(* Logix 5000 project; controller cal1615 1756-L62 rev 20.11; software revision 20.05; part 51 of 82 *)
(* tags used below, declared in another part *)
   FAULT : BOOL;   // Fault AFI
   HMI : BOOL;   // AFI HMI
   p01r09_pb_global_reset : BOOL;   // System Modes PB: Global Fault Reset
   p23_ai_os_gap_dint : DINT;
   p23_ai_os_masked_gap : REAL;
   p23_ai_servo_os_position : REAL;   // Impreg Inputs Servo Operator Side Position
   p23_ai_servo_os_torque : REAL;   // Impreg Inputs Servo Operator Side Torque
   p23_ao_selected_speed : REAL;   // Impreg Metering Roll VFD Selected Speed
   p23_ao_servo_ds_jog_vel_cmd : REAL;   // Impreg Servo Drive Side Jog Velocity Command [in/sec]
   p23_ao_servo_ds_position_cmd : REAL;   // Impreg Servo Drive Side Position Command
   p23_ao_servo_ds_velocity_cmd : REAL;   // Impreg Servo Drive Side Velocity Command
   p23_ao_servo_ds_zero_offset : REAL;   // Impreg Analog Outputs Drive Side Servo Position Offset
   p23_ao_servo_os_jog_vel_cmd : REAL;   // Impreg Servo Operator Side Jog Velocity Command [in/sec]
   p23_ao_servo_os_position_cmd : REAL;   // Impreg Servo Operator Side Position Command
   p23_ao_servo_os_velocity_cmd : REAL;   // Impreg Servo Operator Side Velocity Command
   p23_ao_servo_os_zero_offset : REAL;   // Impreg Analog Outputs Drive Operator Side Servo Position Offset
   p23_ao_supply_selected_speed : REAL;   // Impreg Supply VFD Selected Speed
   p23_cpr_gear_ratio : REAL;
   p23_cpr_roll_diameter_ft : REAL;
   p23_cpr_speed_to_vfd : SYS_SPEED_TO_VFD;   // Impreg Outputs Speed to Impreg Pick Up Roll VFD
   p23_di_impreg_tank_up : BOOL;   // Input Impreg Dip Tank Up
   p23_di_metering_roll : acs800_di_normal;   // Impreg Digital Inputs Metering Roll VFD
   p23_di_servo_ds : servo_di;   // Impreg Digital Inputs Servo Drive Side
   p23_di_servo_os : servo_di;   // Impreg Digital Inputs Servo Operator Side
   p23_di_supply : acs800_di_normal;   // Impreg Supply VFD VFD Inputs
   p23_di_tank_level_high : BOOL;   // Impreg Input Dip Impreg Level High
   p23_di_tank_level_low : BOOL;   // Impreg Input Dip Impreg Level Low
   p23_di_though_level_low : BOOL;   // Impreg Input Dip Impreg Through Level Low
   p23_dint_to_hmi : DINT[17];   // Impreg Dint to HMI
   p23_do_enable_impreg_exhaust_fan : BOOL;   // Impreg Enclosure Digital Output Exhaust Fan Enable
   p23_do_enable_impreg_supply_fan : BOOL;   // Impreg Enclosure Digital Output Supply Fan Enable
   p23_do_impreg : acs800_do_normal;   // Impreg Digital Outputs VFD
   p23_do_impreg_nip_close : BOOL;   // Impreg Digital Output Impreg Nip close
   p23_do_servo_ds : servo_do;   // Impreg Digital Outputs Drive Side Servo
   p23_do_servo_os : servo_do;   // Impreg Digital Outputs Operator Side Servo
   p23_do_Spring : acs800_do_normal;
   p23_do_supply : acs800_do_normal;   // Impreg Supply VFD] Outputs
   p23_servo_ds_error : SYS_ENC_WITH_ZERO_BIT;   // Impreg Dint to HMI Servo Drive Side Error
   p23_servo_ds_warning : SYS_ENC_WITH_ZERO_BIT;   // Impreg Dint to HMI Servo Drive Side Warning
   p23_servo_os_error : SYS_ENC_WITH_ZERO_BIT;   // Impreg Dint to HMI Servo Operator Side Error
   p23_spring_gear_ratio : REAL;
   p23_spring_roll_diameter_ft : REAL;
   p23_spring_speed_to_vfd : SYS_SPEED_TO_VFD;
   p23r01 : routine;   // Impreg Main
   p23r03 : routine;   // Impreg Inputs
   p23r03_timer_fault : TIMER[4];   // Impreg Inputs Timer Fault
   p23r03_timer_warning : TIMER[4];   // Impreg Inputs Timer Warning
   p23r04 : routine;   // Impreg Outputs
   p23r04_timer_fault : TIMER[4];   // Impreg Outputs Fault Delay
   p23r04_timer_warning : TIMER[4];   // Impreg Outputs Warning Delay
   p23r05 : routine;   // Impreg Dint to HMI
   p23r11_servo_not_ready : BOOL;   // Impreg Servo Operator Side Not Ready
   p23r11_servo_status_ab : BOOL;   // Impreg Servo Operator Side AB Status
   p23r11_servo_status_af : BOOL;   // Impreg Servo Operator Side AF Status
   p23r11_servo_status_bb : BOOL;   // Impreg Servo Operator Side BB Status
   p23r12_servo_not_ready : BOOL;   // Impreg Servo Drive Side Not Ready
   p23r12_servo_status_ab : BOOL;   // Impreg Servo Drive Side AB Status
   p23r12_servo_status_af : BOOL;   // Impreg Servo Drive Side AF Status
   p23r12_servo_status_bb : BOOL;   // Impreg Servo Drive Side BB Status
   p23r15_pid_tension_control : BOOL;   // Impreg Metering Roll VFD PID Wet Web Active
   p23r17_adjusted_speed : REAL;
(* P23_Impreg, continued *)

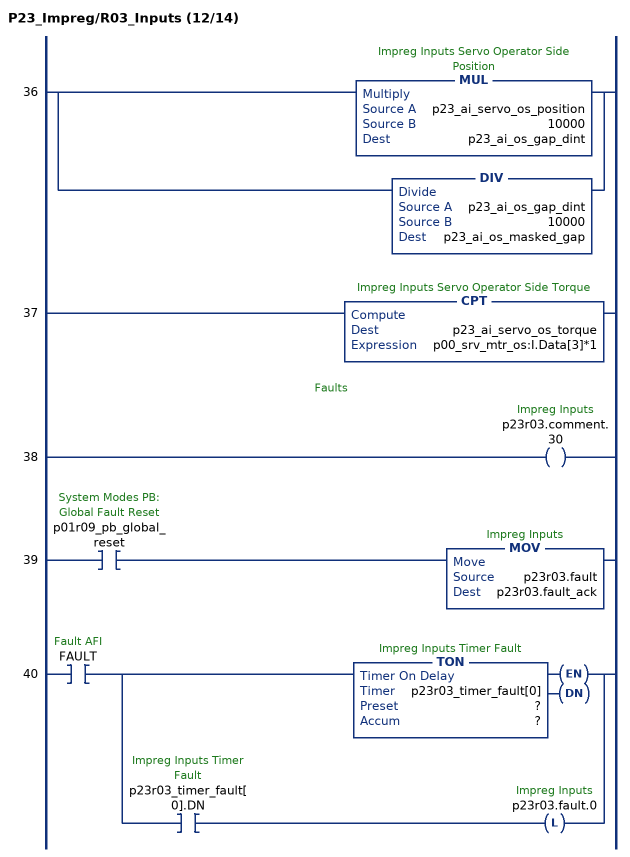
   [picture p993: P23_Impreg/R03_Inputs rungs 36-40]
   36: [MUL(p23_ai_servo_os_position,10000,p23_ai_os_gap_dint) ,DIV(p23_ai_os_gap_dint,10000,p23_ai_os_masked_gap) ];
   37: CPT(p23_ai_servo_os_torque,p00_srv_mtr_os:I.Data[3]*1);
   // Faults
   38: OTE(p23r03.comment.30);
   39: XIC(p01r09_pb_global_reset)MOV(p23r03.fault,p23r03.fault_ack);
   40: XIC(FAULT)[TON(p23r03_timer_fault[0],?,?) ,XIC(p23r03_timer_fault[0].DN) OTL(p23r03.fault.0) ];
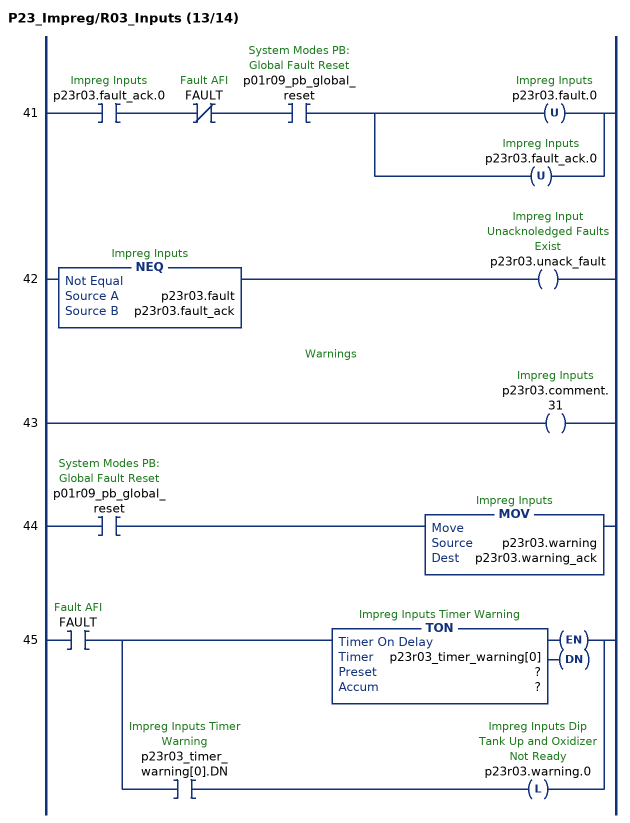
   41: XIC(p23r03.fault_ack.0)XIO(FAULT)XIC(p01r09_pb_global_reset)[OTU(p23r03.fault.0) ,OTU(p23r03.fault_ack.0) ];
   42: NEQ(p23r03.fault,p23r03.fault_ack)OTE(p23r03.unack_fault);
   // Warnings
   43: OTE(p23r03.comment.31);
   44: XIC(p01r09_pb_global_reset)MOV(p23r03.warning,p23r03.warning_ack);
   45: XIC(FAULT)[TON(p23r03_timer_warning[0],?,?) ,XIC(p23r03_timer_warning[0].DN) OTL(p23r03.warning.0) ];
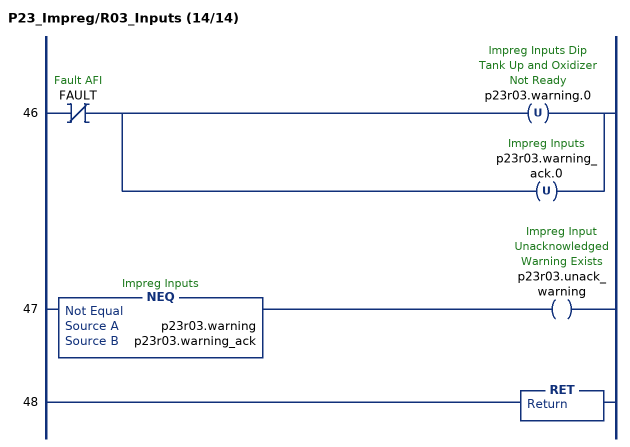
   46: XIO(FAULT)[OTU(p23r03.warning.0) ,OTU(p23r03.warning_ack.0) ];
   47: NEQ(p23r03.warning,p23r03.warning_ack)OTE(p23r03.unack_warning);
   48: RET();
END_ROUTINE

ROUTINE R04_Outputs   (* ladder *)
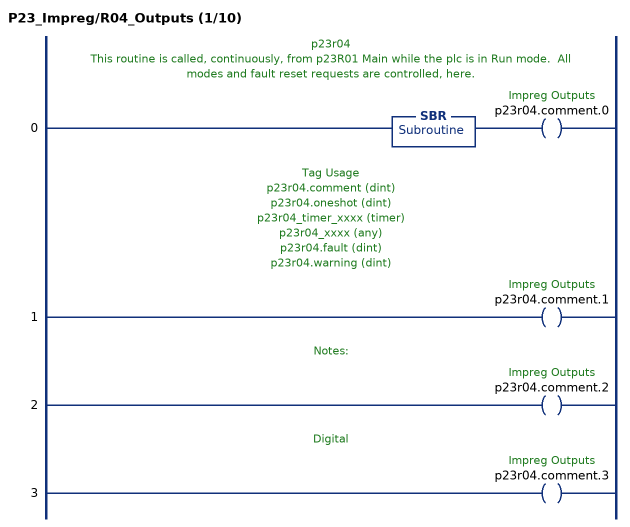
   // p23r04
   // This routine is called, continuously, from p23R01 Main while the plc is in Run mode.  All modes and fault reset requests are controlled, here.
   0: SBR()OTE(p23r04.comment.0);
   // Tag Usage
   // p23r04.comment (dint)
   // p23r04.oneshot (dint)
   // p23r04_timer_xxxx (timer)
   // p23r04_xxxx (any)
   // p23r04.fault (dint)
   // p23r04.warning (dint)
   1: OTE(p23r04.comment.1);
   // Notes:
   2: OTE(p23r04.comment.2);
   // Digital
   3: OTE(p23r04.comment.3);
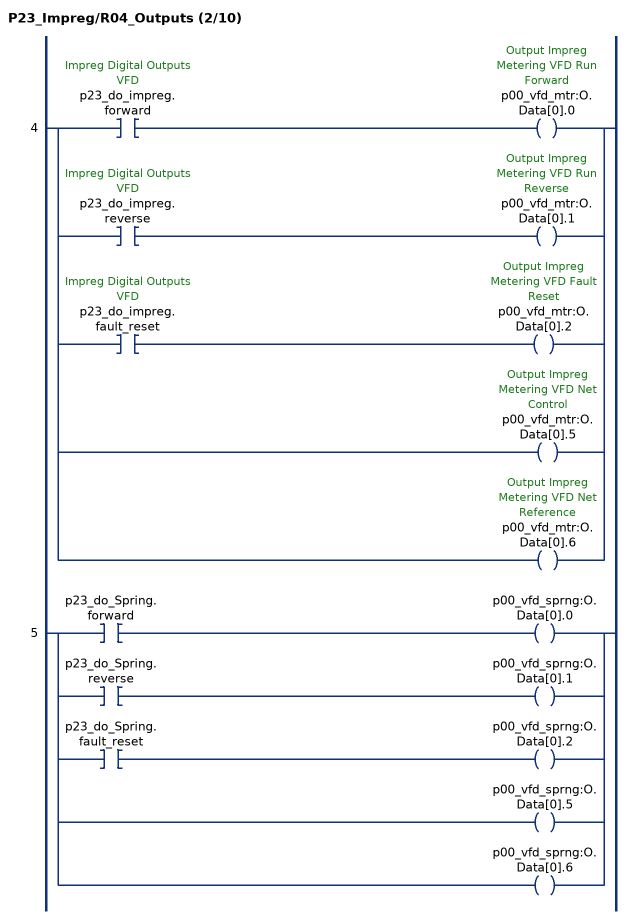
   4: [XIC(p23_do_impreg.forward) OTE(p00_vfd_mtr:O.Data[0].0) ,XIC(p23_do_impreg.reverse) OTE(p00_vfd_mtr:O.Data[0].1) ,XIC(p23_do_impreg.fault_reset) OTE(p00_vfd_mtr:O.Data[0].2) ,OTE(p00_vfd_mtr:O.Data[0].5) ,OTE(p00_vfd_mtr:O.Data[0].6) ];
   5: [XIC(p23_do_Spring.forward) OTE(p00_vfd_sprng:O.Data[0].0) ,XIC(p23_do_Spring.reverse) OTE(p00_vfd_sprng:O.Data[0].1) ,XIC(p23_do_Spring.fault_reset) OTE(p00_vfd_sprng:O.Data[0].2) ,OTE(p00_vfd_sprng:O.Data[0].5) ,OTE(p00_vfd_sprng:O.Data[0].6) ];
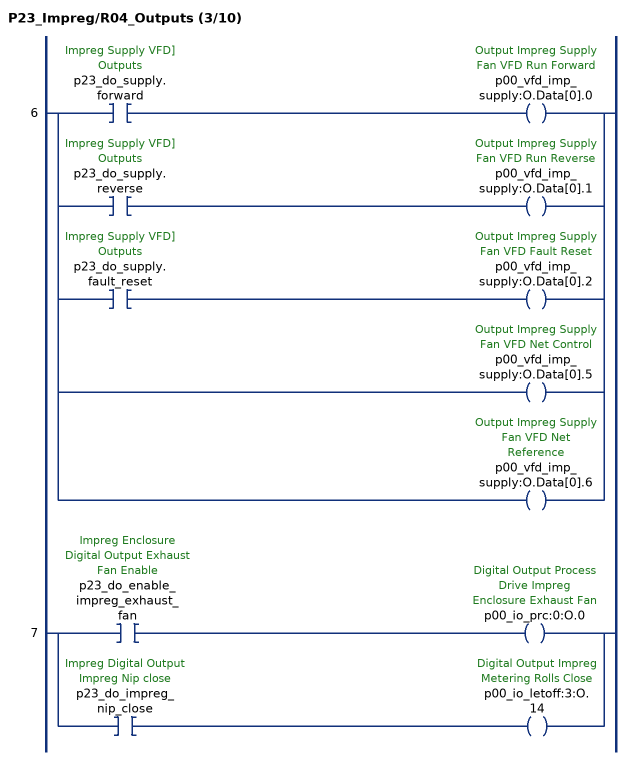
   6: [XIC(p23_do_supply.forward) OTE(p00_vfd_imp_supply:O.Data[0].0) ,XIC(p23_do_supply.reverse) OTE(p00_vfd_imp_supply:O.Data[0].1) ,XIC(p23_do_supply.fault_reset) OTE(p00_vfd_imp_supply:O.Data[0].2) ,OTE(p00_vfd_imp_supply:O.Data[0].5) ,OTE(p00_vfd_imp_supply:O.Data[0].6) ];
   7: [XIC(p23_do_enable_impreg_exhaust_fan) OTE(p00_io_prc:0:O.0) ,XIC(p23_do_impreg_nip_close) OTE(p00_io_letoff:3:O.14) ];
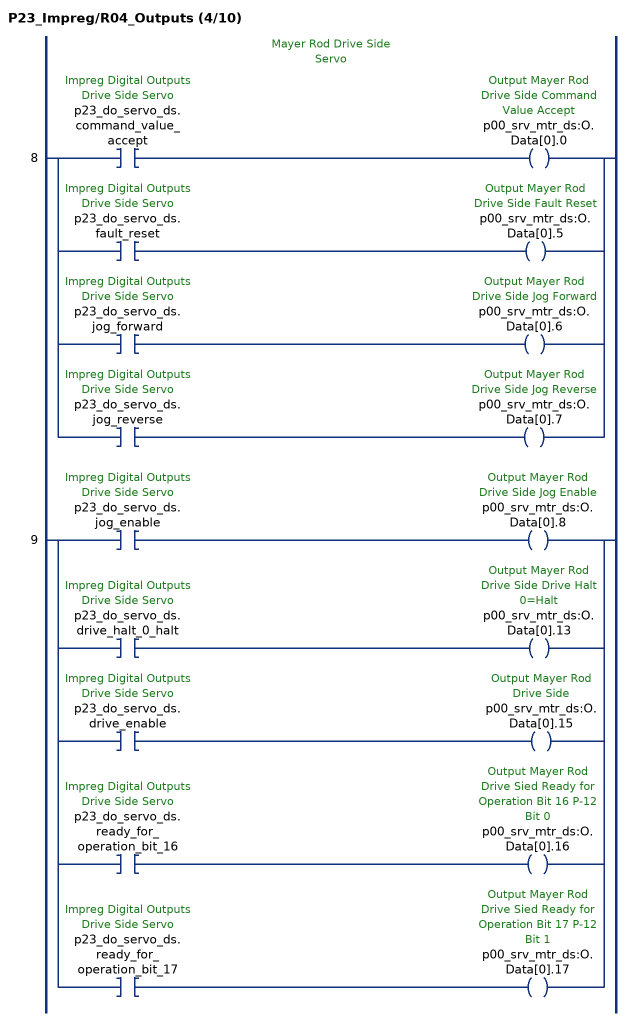
   // Mayer Rod Drive Side
   // Servo
   8: [XIC(p23_do_servo_ds.command_value_accept) OTE(p00_srv_mtr_ds:O.Data[0].0) ,XIC(p23_do_servo_ds.fault_reset) OTE(p00_srv_mtr_ds:O.Data[0].5) ,XIC(p23_do_servo_ds.jog_forward) OTE(p00_srv_mtr_ds:O.Data[0].6) ,XIC(p23_do_servo_ds.jog_reverse) OTE(p00_srv_mtr_ds:O.Data[0].7) ];
   9: [XIC(p23_do_servo_ds.jog_enable) OTE(p00_srv_mtr_ds:O.Data[0].8) ,XIC(p23_do_servo_ds.drive_halt_0_halt) OTE(p00_srv_mtr_ds:O.Data[0].13) ,XIC(p23_do_servo_ds.drive_enable) OTE(p00_srv_mtr_ds:O.Data[0].15) ,XIC(p23_do_servo_ds.ready_for_operation_bit_16) OTE(p00_srv_mtr_ds:O.Data[0].16) ,XIC(p23_do_servo_ds.ready_for_operation_bit_17) OTE(p00_srv_mtr_ds:O.Data[0].17) ];
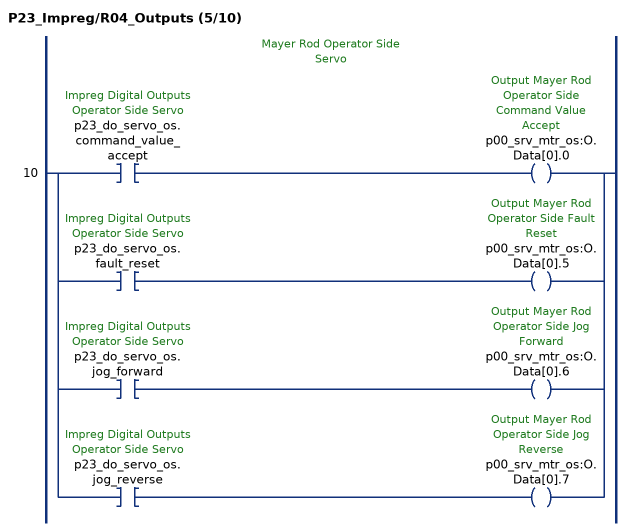
   // Mayer Rod Operator Side
   // Servo
   10: [XIC(p23_do_servo_os.command_value_accept) OTE(p00_srv_mtr_os:O.Data[0].0) ,XIC(p23_do_servo_os.fault_reset) OTE(p00_srv_mtr_os:O.Data[0].5) ,XIC(p23_do_servo_os.jog_forward) OTE(p00_srv_mtr_os:O.Data[0].6) ,XIC(p23_do_servo_os.jog_reverse) OTE(p00_srv_mtr_os:O.Data[0].7) ];
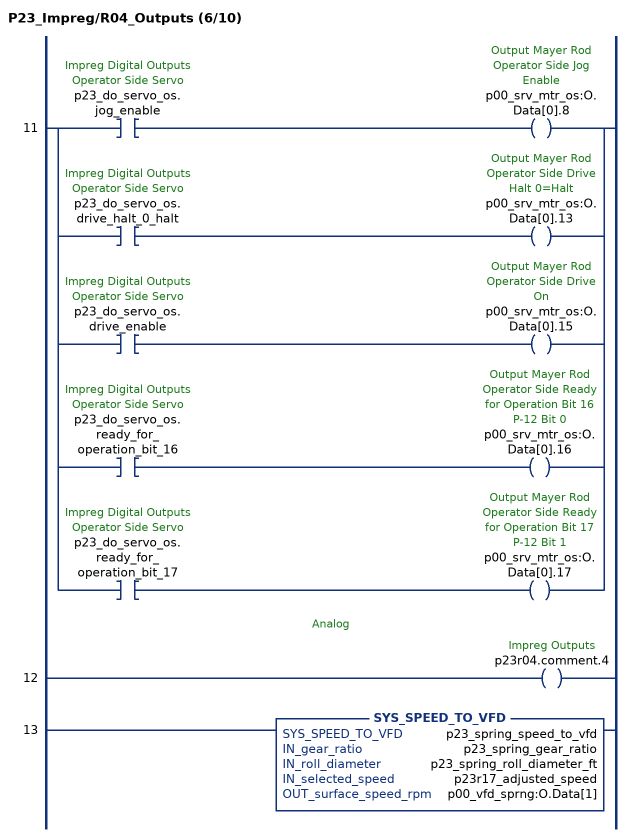
   11: [XIC(p23_do_servo_os.jog_enable) OTE(p00_srv_mtr_os:O.Data[0].8) ,XIC(p23_do_servo_os.drive_halt_0_halt) OTE(p00_srv_mtr_os:O.Data[0].13) ,XIC(p23_do_servo_os.drive_enable) OTE(p00_srv_mtr_os:O.Data[0].15) ,XIC(p23_do_servo_os.ready_for_operation_bit_16) OTE(p00_srv_mtr_os:O.Data[0].16) ,XIC(p23_do_servo_os.ready_for_operation_bit_17) OTE(p00_srv_mtr_os:O.Data[0].17) ];
   // Analog
   12: OTE(p23r04.comment.4);
   13: SYS_SPEED_TO_VFD(p23_spring_speed_to_vfd,p23_spring_gear_ratio,p23_spring_roll_diameter_ft,p23r17_adjusted_speed,p00_vfd_sprng:O.Data[1]);
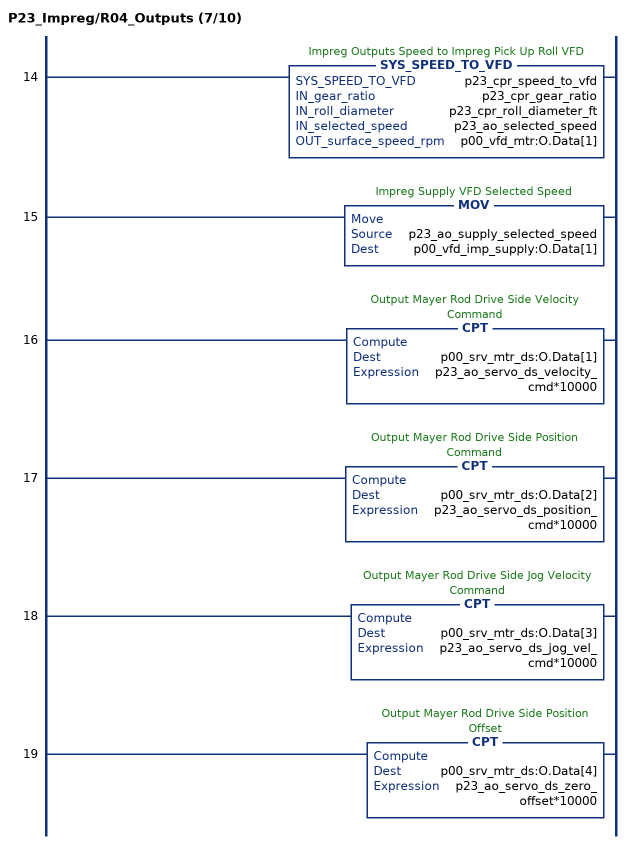
   14: SYS_SPEED_TO_VFD(p23_cpr_speed_to_vfd,p23_cpr_gear_ratio,p23_cpr_roll_diameter_ft,p23_ao_selected_speed,p00_vfd_mtr:O.Data[1]);
   15: MOV(p23_ao_supply_selected_speed,p00_vfd_imp_supply:O.Data[1]);
   16: CPT(p00_srv_mtr_ds:O.Data[1],p23_ao_servo_ds_velocity_cmd*10000);
   17: CPT(p00_srv_mtr_ds:O.Data[2],p23_ao_servo_ds_position_cmd*10000);
   18: CPT(p00_srv_mtr_ds:O.Data[3],p23_ao_servo_ds_jog_vel_cmd*10000);
   19: CPT(p00_srv_mtr_ds:O.Data[4],p23_ao_servo_ds_zero_offset*10000);
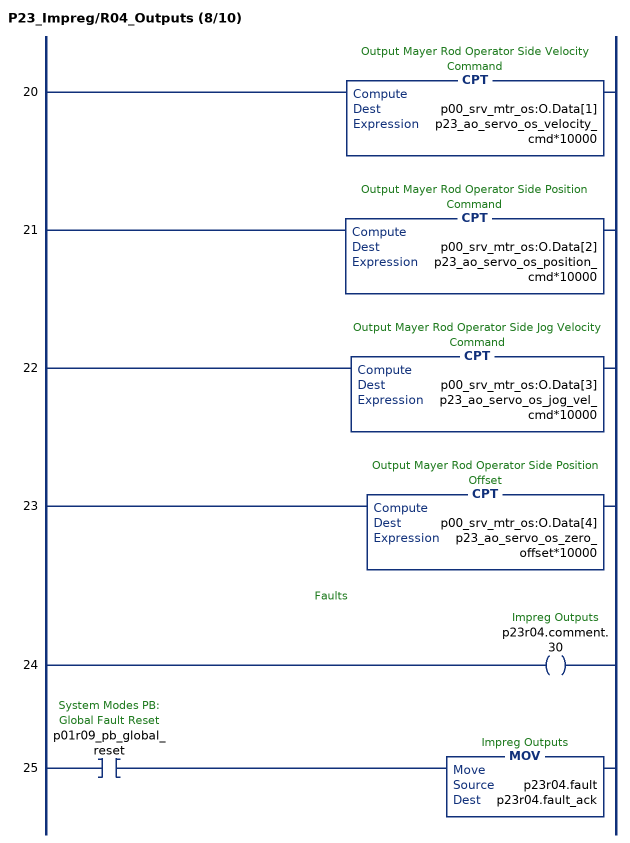
   20: CPT(p00_srv_mtr_os:O.Data[1],p23_ao_servo_os_velocity_cmd*10000);
   21: CPT(p00_srv_mtr_os:O.Data[2],p23_ao_servo_os_position_cmd*10000);
   22: CPT(p00_srv_mtr_os:O.Data[3],p23_ao_servo_os_jog_vel_cmd*10000);
   23: CPT(p00_srv_mtr_os:O.Data[4],p23_ao_servo_os_zero_offset*10000);
   // Faults
   24: OTE(p23r04.comment.30);
   25: XIC(p01r09_pb_global_reset)MOV(p23r04.fault,p23r04.fault_ack);
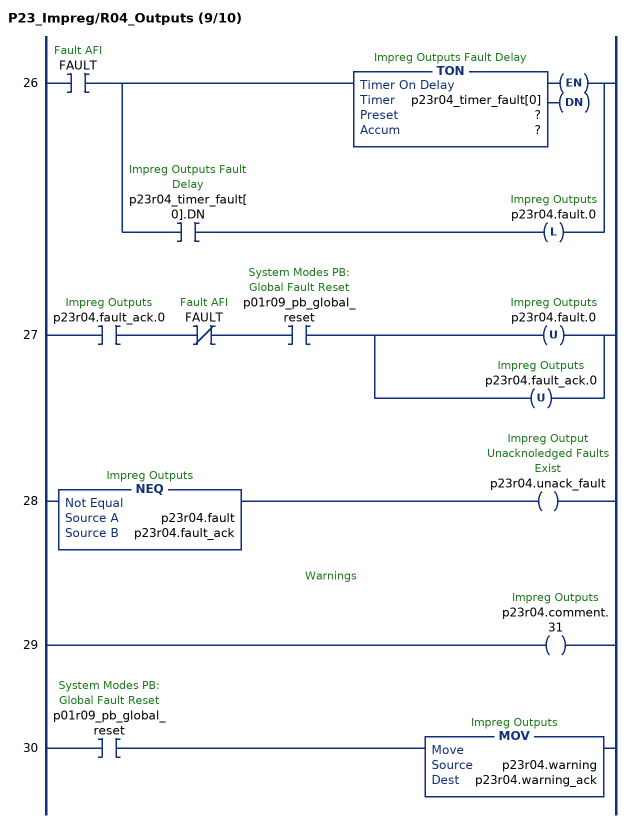
   26: XIC(FAULT)[TON(p23r04_timer_fault[0],?,?) ,XIC(p23r04_timer_fault[0].DN) OTL(p23r04.fault.0) ];
   27: XIC(p23r04.fault_ack.0)XIO(FAULT)XIC(p01r09_pb_global_reset)[OTU(p23r04.fault.0) ,OTU(p23r04.fault_ack.0) ];
   28: NEQ(p23r04.fault,p23r04.fault_ack)OTE(p23r04.unack_fault);
   // Warnings
   29: OTE(p23r04.comment.31);
   30: XIC(p01r09_pb_global_reset)MOV(p23r04.warning,p23r04.warning_ack);
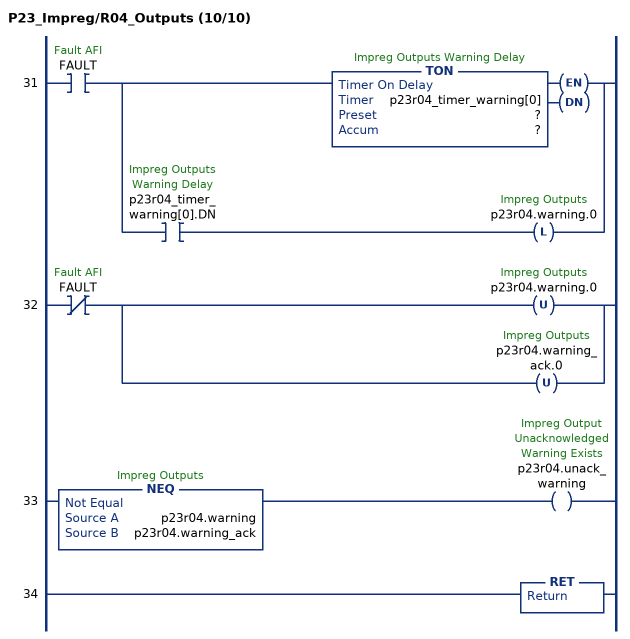
   31: XIC(FAULT)[TON(p23r04_timer_warning[0],?,?) ,XIC(p23r04_timer_warning[0].DN) OTL(p23r04.warning.0) ];
   32: XIO(FAULT)[OTU(p23r04.warning.0) ,OTU(p23r04.warning_ack.0) ];
   33: NEQ(p23r04.warning,p23r04.warning_ack)OTE(p23r04.unack_warning);
   34: RET();
END_ROUTINE

ROUTINE R05_Dint_to_HMI   (* ladder *)
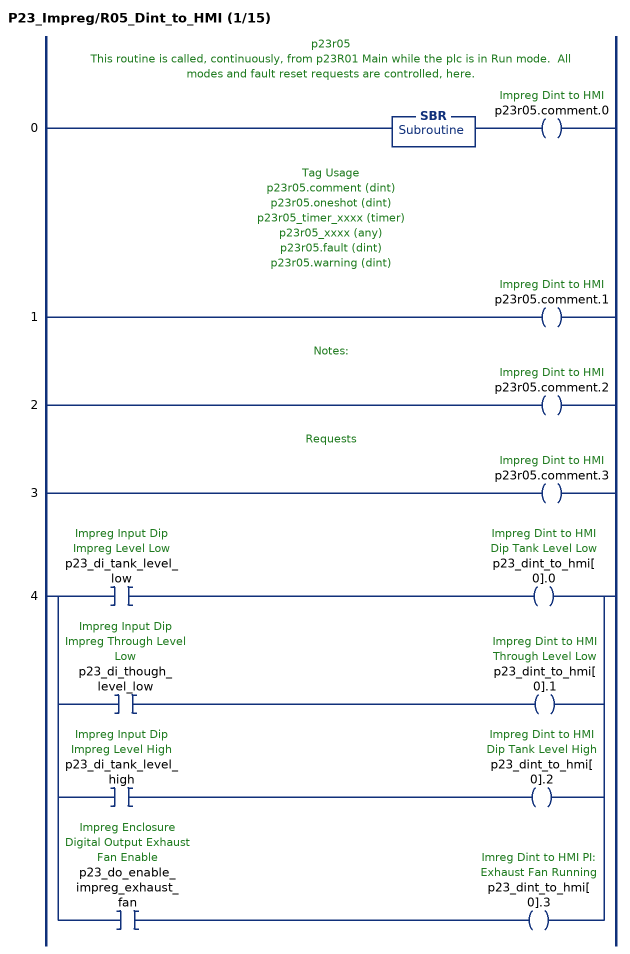
   // p23r05
   // This routine is called, continuously, from p23R01 Main while the plc is in Run mode.  All modes and fault reset requests are controlled, here.
   0: SBR()OTE(p23r05.comment.0);
   // Tag Usage
   // p23r05.comment (dint)
   // p23r05.oneshot (dint)
   // p23r05_timer_xxxx (timer)
   // p23r05_xxxx (any)
   // p23r05.fault (dint)
   // p23r05.warning (dint)
   1: OTE(p23r05.comment.1);
   // Notes:
   2: OTE(p23r05.comment.2);
   // Requests
   3: OTE(p23r05.comment.3);
   4: [XIC(p23_di_tank_level_low) OTE(p23_dint_to_hmi[0].0) ,XIC(p23_di_though_level_low) OTE(p23_dint_to_hmi[0].1) ,XIC(p23_di_tank_level_high) OTE(p23_dint_to_hmi[0].2) ,XIC(p23_do_enable_impreg_exhaust_fan) OTE(p23_dint_to_hmi[0].3) ];
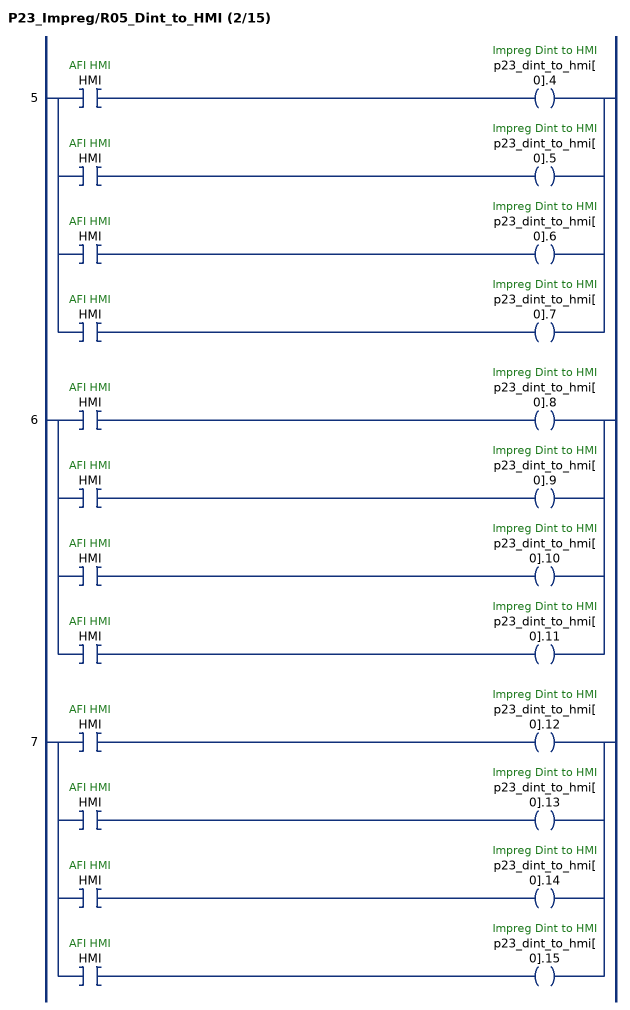
   5: [XIC(HMI) OTE(p23_dint_to_hmi[0].4) ,XIC(HMI) OTE(p23_dint_to_hmi[0].5) ,XIC(HMI) OTE(p23_dint_to_hmi[0].6) ,XIC(HMI) OTE(p23_dint_to_hmi[0].7) ];
   6: [XIC(HMI) OTE(p23_dint_to_hmi[0].8) ,XIC(HMI) OTE(p23_dint_to_hmi[0].9) ,XIC(HMI) OTE(p23_dint_to_hmi[0].10) ,XIC(HMI) OTE(p23_dint_to_hmi[0].11) ];
   7: [XIC(HMI) OTE(p23_dint_to_hmi[0].12) ,XIC(HMI) OTE(p23_dint_to_hmi[0].13) ,XIC(HMI) OTE(p23_dint_to_hmi[0].14) ,XIC(HMI) OTE(p23_dint_to_hmi[0].15) ];
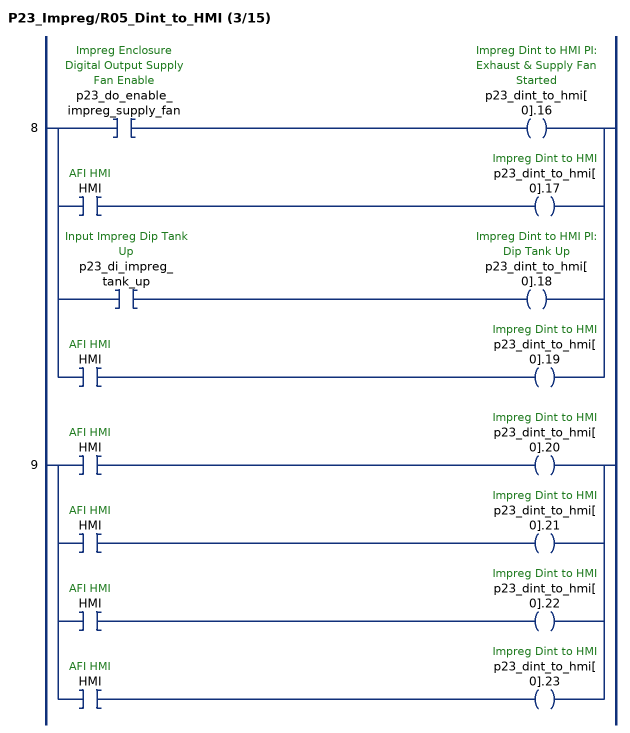
   8: [XIC(p23_do_enable_impreg_supply_fan) OTE(p23_dint_to_hmi[0].16) ,XIC(HMI) OTE(p23_dint_to_hmi[0].17) ,XIC(p23_di_impreg_tank_up) OTE(p23_dint_to_hmi[0].18) ,XIC(HMI) OTE(p23_dint_to_hmi[0].19) ];
   9: [XIC(HMI) OTE(p23_dint_to_hmi[0].20) ,XIC(HMI) OTE(p23_dint_to_hmi[0].21) ,XIC(HMI) OTE(p23_dint_to_hmi[0].22) ,XIC(HMI) OTE(p23_dint_to_hmi[0].23) ];
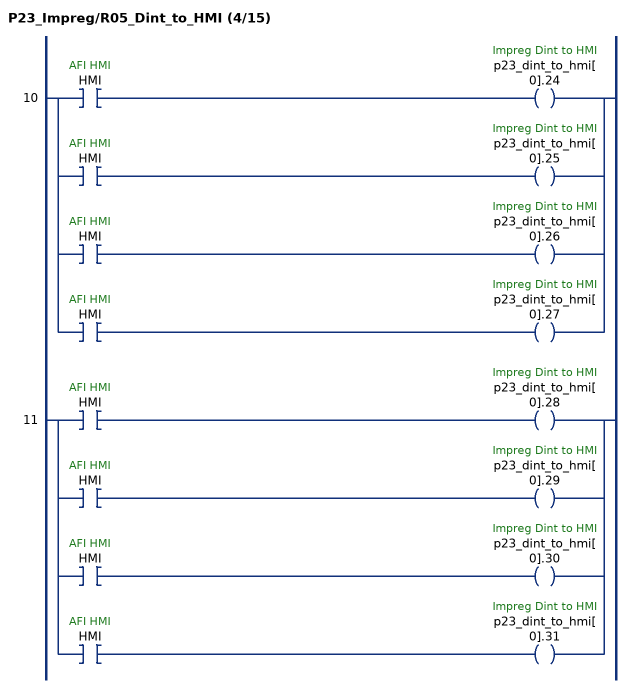
   10: [XIC(HMI) OTE(p23_dint_to_hmi[0].24) ,XIC(HMI) OTE(p23_dint_to_hmi[0].25) ,XIC(HMI) OTE(p23_dint_to_hmi[0].26) ,XIC(HMI) OTE(p23_dint_to_hmi[0].27) ];
   11: [XIC(HMI) OTE(p23_dint_to_hmi[0].28) ,XIC(HMI) OTE(p23_dint_to_hmi[0].29) ,XIC(HMI) OTE(p23_dint_to_hmi[0].30) ,XIC(HMI) OTE(p23_dint_to_hmi[0].31) ];
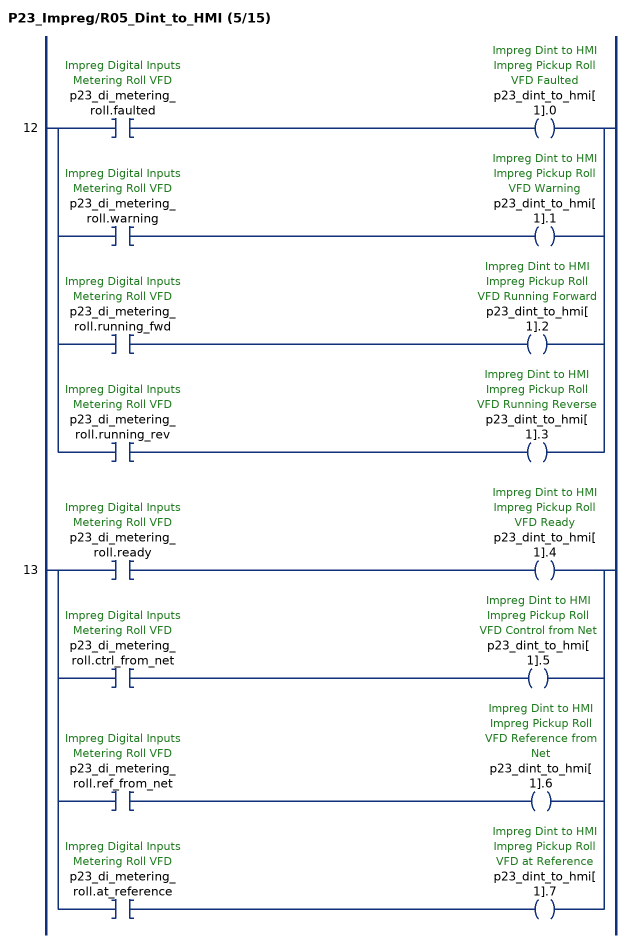
   12: [XIC(p23_di_metering_roll.faulted) OTE(p23_dint_to_hmi[1].0) ,XIC(p23_di_metering_roll.warning) OTE(p23_dint_to_hmi[1].1) ,XIC(p23_di_metering_roll.running_fwd) OTE(p23_dint_to_hmi[1].2) ,XIC(p23_di_metering_roll.running_rev) OTE(p23_dint_to_hmi[1].3) ];
   13: [XIC(p23_di_metering_roll.ready) OTE(p23_dint_to_hmi[1].4) ,XIC(p23_di_metering_roll.ctrl_from_net) OTE(p23_dint_to_hmi[1].5) ,XIC(p23_di_metering_roll.ref_from_net) OTE(p23_dint_to_hmi[1].6) ,XIC(p23_di_metering_roll.at_reference) OTE(p23_dint_to_hmi[1].7) ];
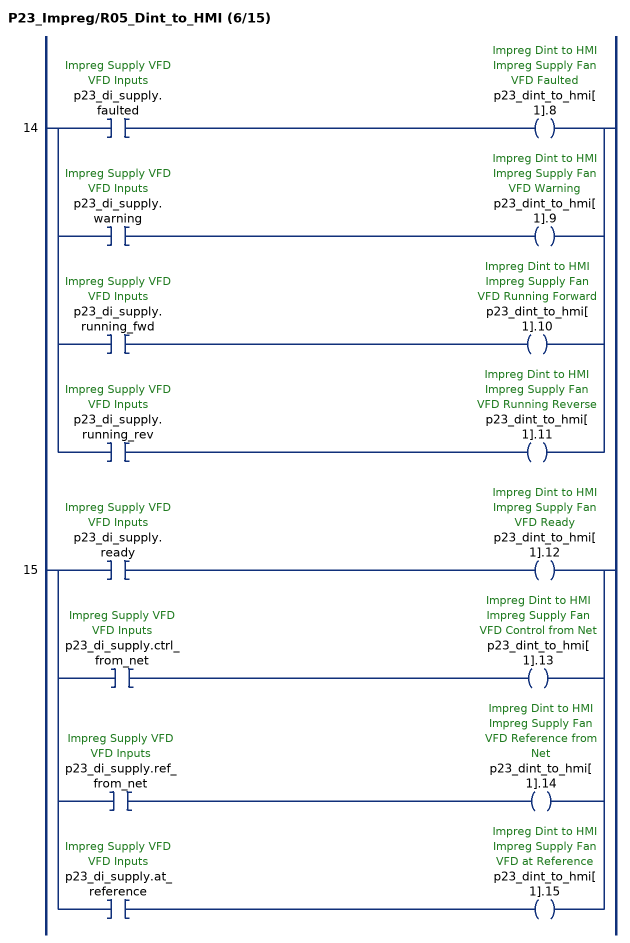
   14: [XIC(p23_di_supply.faulted) OTE(p23_dint_to_hmi[1].8) ,XIC(p23_di_supply.warning) OTE(p23_dint_to_hmi[1].9) ,XIC(p23_di_supply.running_fwd) OTE(p23_dint_to_hmi[1].10) ,XIC(p23_di_supply.running_rev) OTE(p23_dint_to_hmi[1].11) ];
   15: [XIC(p23_di_supply.ready) OTE(p23_dint_to_hmi[1].12) ,XIC(p23_di_supply.ctrl_from_net) OTE(p23_dint_to_hmi[1].13) ,XIC(p23_di_supply.ref_from_net) OTE(p23_dint_to_hmi[1].14) ,XIC(p23_di_supply.at_reference) OTE(p23_dint_to_hmi[1].15) ];
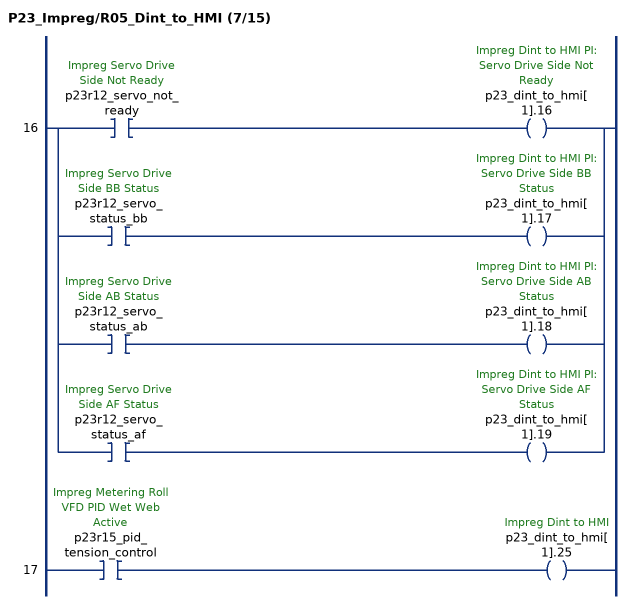
   16: [XIC(p23r12_servo_not_ready) OTE(p23_dint_to_hmi[1].16) ,XIC(p23r12_servo_status_bb) OTE(p23_dint_to_hmi[1].17) ,XIC(p23r12_servo_status_ab) OTE(p23_dint_to_hmi[1].18) ,XIC(p23r12_servo_status_af) OTE(p23_dint_to_hmi[1].19) ];
   17: XIC(p23r15_pid_tension_control)OTE(p23_dint_to_hmi[1].25);
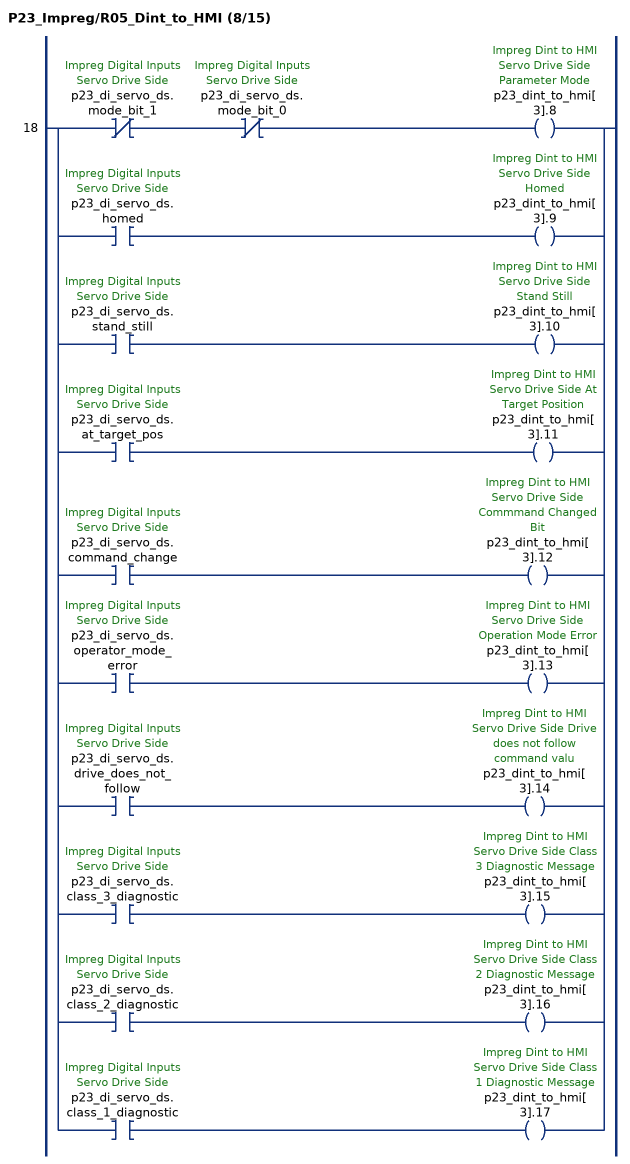
   18: [XIO(p23_di_servo_ds.mode_bit_1) XIO(p23_di_servo_ds.mode_bit_0) OTE(p23_dint_to_hmi[3].8) ,XIC(p23_di_servo_ds.homed) OTE(p23_dint_to_hmi[3].9) ,XIC(p23_di_servo_ds.stand_still) OTE(p23_dint_to_hmi[3].10) ,XIC(p23_di_servo_ds.at_target_pos) OTE(p23_dint_to_hmi[3].11) ,XIC(p23_di_servo_ds.command_change) OTE(p23_dint_to_hmi[3].12) ,XIC(p23_di_servo_ds.operator_mode_error) OTE(p23_dint_to_hmi[3].13) ,XIC(p23_di_servo_ds.drive_does_not_follow) OTE(p23_dint_to_hmi[3].14) ,XIC(p23_di_servo_ds.class_3_diagnostic) OTE(p23_dint_to_hmi[3].15) ,XIC(p23_di_servo_ds.class_2_diagnostic) OTE(p23_dint_to_hmi[3].16) ,XIC(p23_di_servo_ds.class_1_diagnostic) OTE(p23_dint_to_hmi[3].17) ];
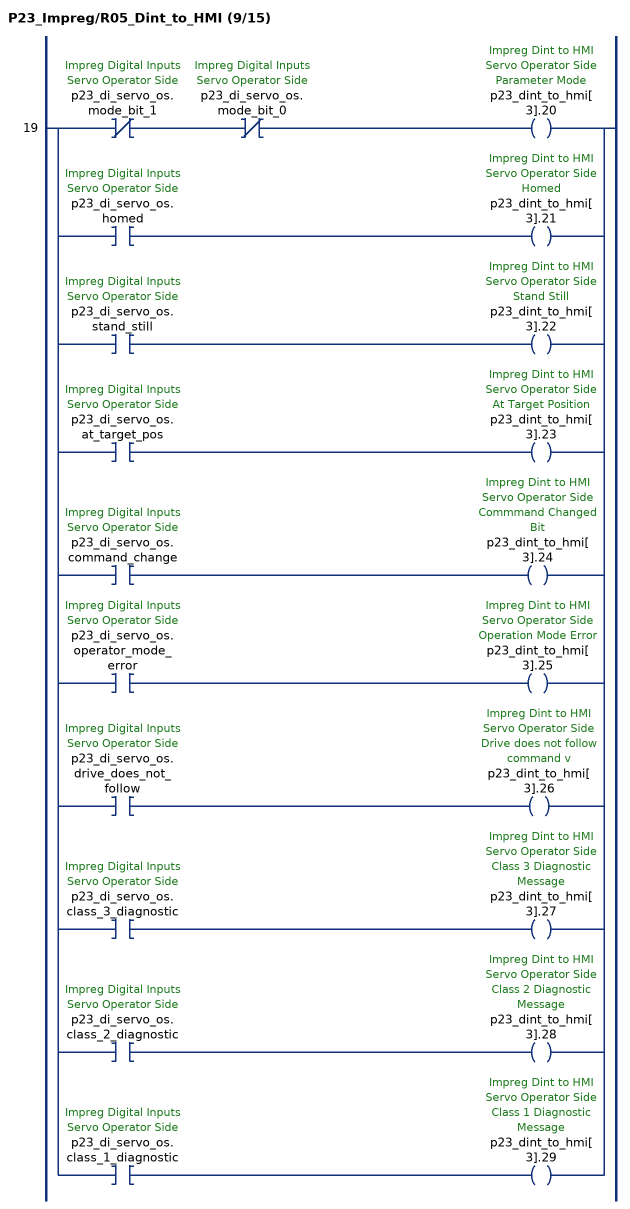
   19: [XIO(p23_di_servo_os.mode_bit_1) XIO(p23_di_servo_os.mode_bit_0) OTE(p23_dint_to_hmi[3].20) ,XIC(p23_di_servo_os.homed) OTE(p23_dint_to_hmi[3].21) ,XIC(p23_di_servo_os.stand_still) OTE(p23_dint_to_hmi[3].22) ,XIC(p23_di_servo_os.at_target_pos) OTE(p23_dint_to_hmi[3].23) ,XIC(p23_di_servo_os.command_change) OTE(p23_dint_to_hmi[3].24) ,XIC(p23_di_servo_os.operator_mode_error) OTE(p23_dint_to_hmi[3].25) ,XIC(p23_di_servo_os.drive_does_not_follow) OTE(p23_dint_to_hmi[3].26) ,XIC(p23_di_servo_os.class_3_diagnostic) OTE(p23_dint_to_hmi[3].27) ,XIC(p23_di_servo_os.class_2_diagnostic) OTE(p23_dint_to_hmi[3].28) ,XIC(p23_di_servo_os.class_1_diagnostic) OTE(p23_dint_to_hmi[3].29) ];
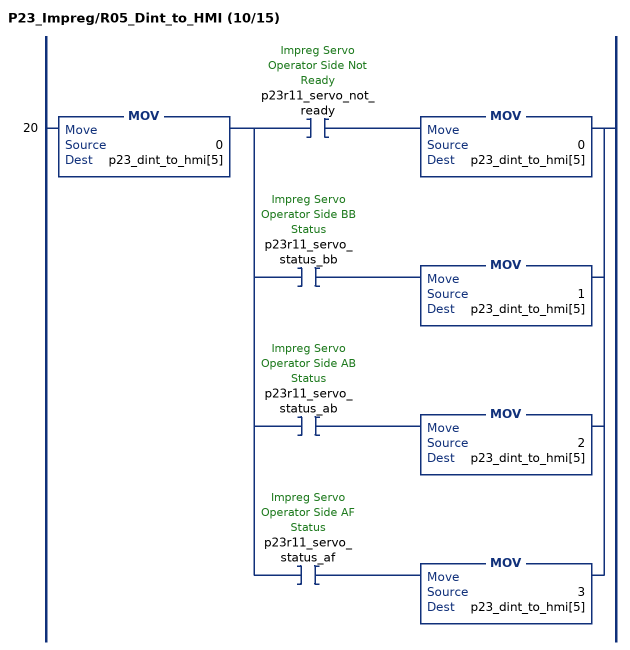
   20: MOV(0,p23_dint_to_hmi[5])[XIC(p23r11_servo_not_ready) MOV(0,p23_dint_to_hmi[5]) ,XIC(p23r11_servo_status_bb) MOV(1,p23_dint_to_hmi[5]) ,XIC(p23r11_servo_status_ab) MOV(2,p23_dint_to_hmi[5]) ,XIC(p23r11_servo_status_af) MOV(3,p23_dint_to_hmi[5]) ];
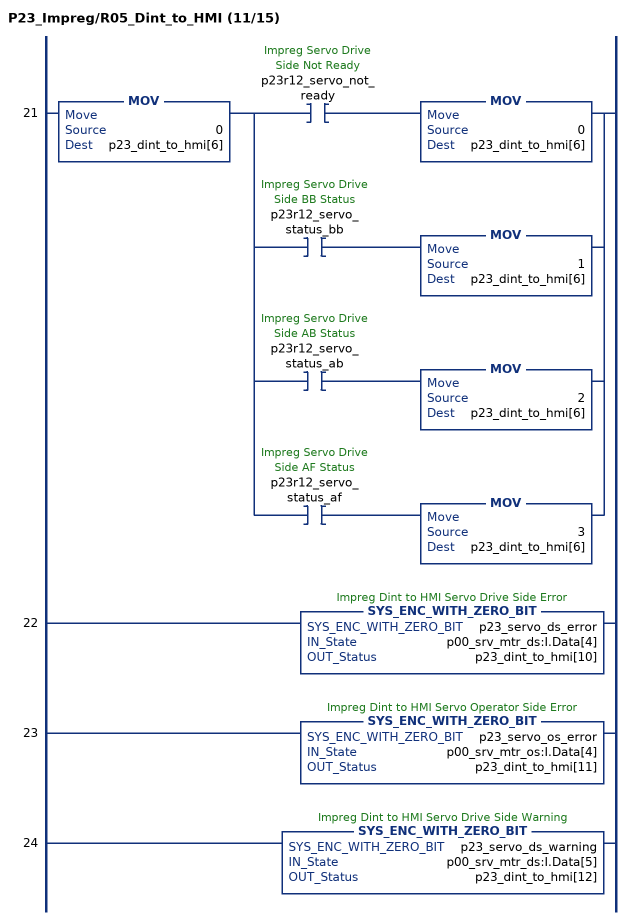
   21: MOV(0,p23_dint_to_hmi[6])[XIC(p23r12_servo_not_ready) MOV(0,p23_dint_to_hmi[6]) ,XIC(p23r12_servo_status_bb) MOV(1,p23_dint_to_hmi[6]) ,XIC(p23r12_servo_status_ab) MOV(2,p23_dint_to_hmi[6]) ,XIC(p23r12_servo_status_af) MOV(3,p23_dint_to_hmi[6]) ];
   22: SYS_ENC_WITH_ZERO_BIT(p23_servo_ds_error,p00_srv_mtr_ds:I.Data[4],p23_dint_to_hmi[10]);
   23: SYS_ENC_WITH_ZERO_BIT(p23_servo_os_error,p00_srv_mtr_os:I.Data[4],p23_dint_to_hmi[11]);
   24: SYS_ENC_WITH_ZERO_BIT(p23_servo_ds_warning,p00_srv_mtr_ds:I.Data[5],p23_dint_to_hmi[12]);
